Staubli VAL3: FC_InitData.pgx

program FC_InitData()
  local num l_ni
  local bool l_bInit
begin
  cls()
  userPage()
  // call hmi_keyinmain()
  bTxt1=false
  bTxt2=false
  bTxt3=false
end
